(* IEC 61131-3 sources: AXOpen/src/inspectors/app/src, 2 files *)

(* ---- configuration.st ---- *)
CONFIGURATION MyConfiguration
    TASK Main(Interval := T#10ms, Priority := 1);
    PROGRAM P1 WITH Main: MyProgram;

    VAR_GLOBAL
        {S7.extern=ReadWrite}
        S71500Rtc :  AXOpen.S71500.Rtc;
        {S7.extern=ReadWrite}
        S71500Rtm :  AXOpen.S71500.Rtm;
        {S7.extern=ReadWrite}
        sandbox : SandboxContext;
        {S7.extern=ReadWrite}
        documentation : DocumentationContext;
    END_VAR
END_CONFIGURATION

(* ---- program.st ---- *)
PROGRAM MyProgram
    VAR_EXTERNAL
        sandbox : SandboxContext;
        documentation : DocumentationContext;
        S71500Rtc :  AXOpen.S71500.Rtc;
        S71500Rtm : AXOpen.S71500.Rtm;
    END_VAR

    VAR

    END_VAR

    VAR_TEMP

    END_VAR
    sandbox.InjectRtc(S71500Rtc);
    sandbox.InjectRtm(S71500Rtm);
    sandbox.Run();

    documentation.InjectRtc(S71500Rtc);
    documentation.InjectRtm(S71500Rtm);
    documentation.Run();
END_PROGRAM
